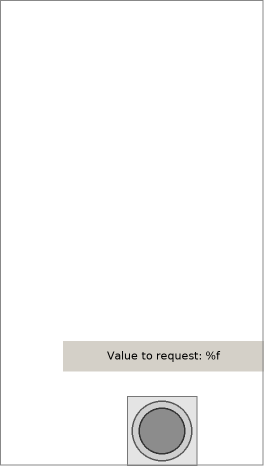
VISUALIZATION Visualization  // 264x466
    Textfield (63,341 201x30), "Value to request: %f", text variable: MAIN.rValueToWrite
        OnMouseClick: write MAIN.rValueToWrite via Default
    PushSwitch (127,396 70x70), variable: MAIN.bRequestToWrite, behaviour: TAP, style: Switch-PushSwitch-Gray
END_VISUALIZATION

(* stored: Version 1.1.0.1, ProductVersion 3.1.4024.12
   Visu Visualization: Id {aab0f211-269d-4d7f-8eea-adeb787c7e10} *)
